FUNCTION_BLOCK HeartBeatSim (* Basic Function Block Type *)
  (* Standard: 61499-2 *)
  (* Version 0.0, 7/17/2026, Schneider Electric, Template *)
  PACKAGE SE.Nereda;
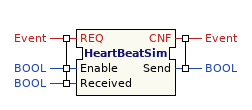
  EVENT_INPUT
    REQ WITH Enable, Received; (* Normal Execution Request *)
  END_EVENT
  EVENT_OUTPUT
    CNF WITH Send; (* Execution Confirmation *)
  END_EVENT
  VAR_INPUT
    Enable : BOOL;
    Received : BOOL;
  END_VAR
  VAR_OUTPUT
    Send : BOOL;
  END_VAR
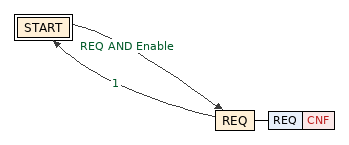
  EC_STATES
    START; (* Initial State *)
    REQ : REQ -> CNF; (* Normal execution *)
  END_STATES
  EC_TRANSITIONS
    START TO REQ := REQ AND Enable;
    REQ TO START := 1;
  END_TRANSITIONS
  ALGORITHM REQ IN ST: (* Normally executed algorithm *)
;
Send := Received;
  END_ALGORITHM
END_FUNCTION_BLOCK
